TYPE ST_PDO_DriveOut :
STRUCT
	SEW_MovidriveControlWord				: ST_MoviDriveCtrlWord;
	ABB_ACS880_ControlWord					: ST_ABBDriveCtrlWord;
	
END_STRUCT
END_TYPE

(* stored: Version 1.1.0.1, ProductVersion 3.1.4022.12
   DUT ST_PDO_DriveOut: Id {1e5c2091-9349-49ea-8053-e226e9ae56e6} *)
